(* PLC project Sin nombre, Desconocido Sin nombre 1 *)
(* stored: creationDateTime 2025-10-27T12:46:01, modificationDateTime 2025-10-27T17:09:16 *)

PROGRAM program0
  VAR
    SensorInclinacion AT %IX0.1 : BOOL;
    SensorFuego AT %IW0 : INT;
    LedAzul AT %QX0.3 : BOOL := FALSE;
    LedParacaidas AT %QX0.4 : BOOL := FALSE;
    LedRojo AT %QX0.1 : BOOL := FALSE;
  END_VAR
  VAR
    EstadoTurbulento : BOOL := FALSE;
    EstadoSobrecalentamiento : BOOL := FALSE;
  END_VAR
  VAR
    LedVerde AT %QX0.2 : BOOL := TRUE;
  END_VAR
  VAR
    EstadoSeguro : BOOL := TRUE;
    UmbralFuego : INT := 1;
    RetardoParacaidas : TIME := T#5000ms;
    Titilo : TIME := T#10ms;
    TiempoSubidaBajada : TIME := T#30000ms;
    RetardoEyeccion : TON;
    AscensoDescenso : TOF;
    ParpadeoLuces : TP;
    Despliegue : TP;
    BiestableAscDesc : RS;
  END_VAR
  VAR  (* added by the conversion: wires and edge detectors of the diagram *)
    _AND42_OUT : BOOL;
    _GT10_OUT : BOOL;
    _AND14_OUT : BOOL;
  END_VAR

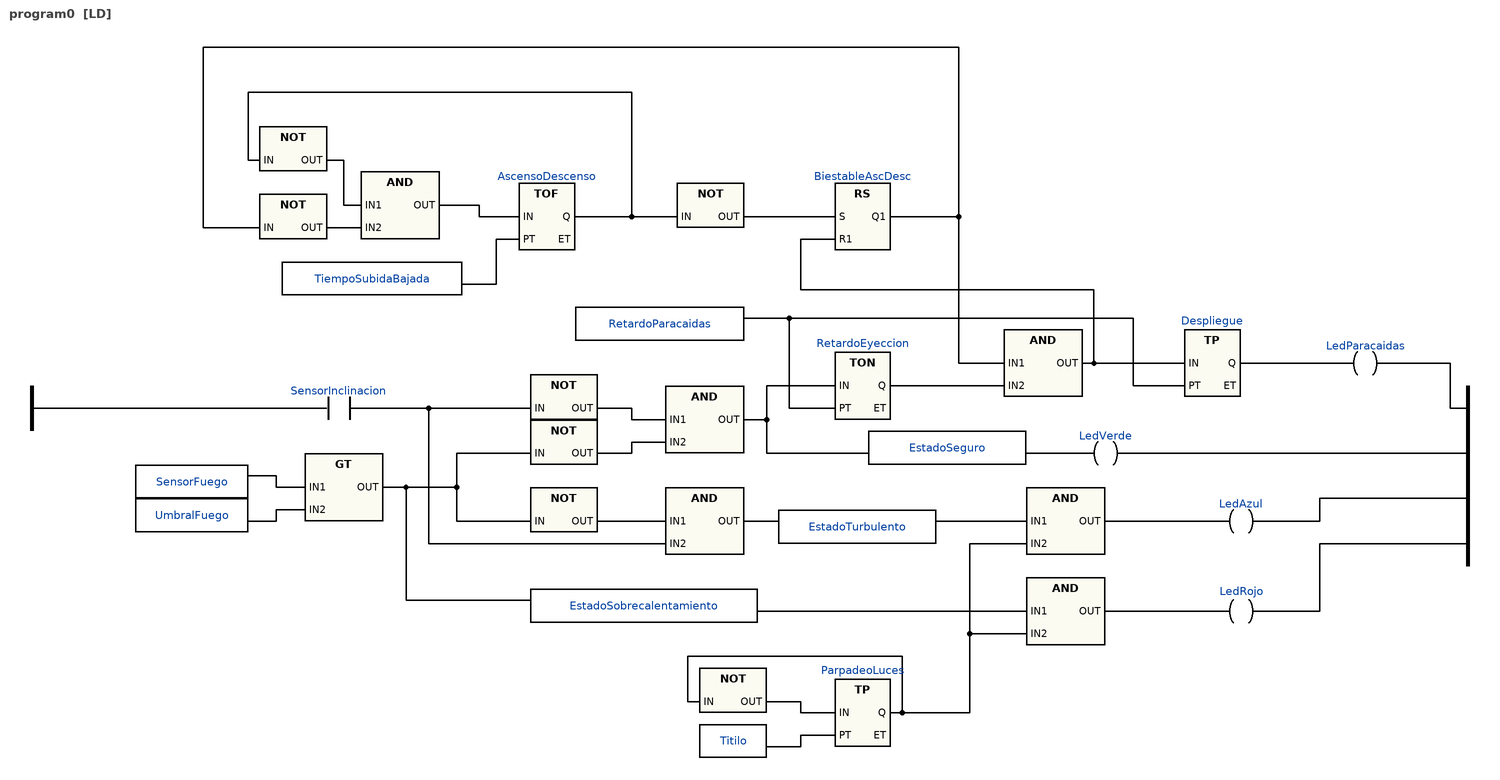
(* LD diagram, written out as Structured Text *)
AscensoDescenso(IN := NOT AscensoDescenso.Q AND NOT BiestableAscDesc.Q1, PT := TiempoSubidaBajada);
BiestableAscDesc(S := NOT AscensoDescenso.Q, R1 := _AND42_OUT);
_GT10_OUT := SensorFuego > UmbralFuego;
_AND14_OUT := NOT SensorInclinacion AND NOT _GT10_OUT;
RetardoEyeccion(IN := _AND14_OUT, PT := RetardoParacaidas);
_AND42_OUT := BiestableAscDesc.Q1 AND RetardoEyeccion.Q;
Despliegue(IN := _AND42_OUT, PT := RetardoParacaidas);
LedParacaidas := Despliegue.Q;
LedVerde := EstadoSeguro;
ParpadeoLuces(IN := NOT ParpadeoLuces.Q, PT := Titilo);
LedAzul := EstadoTurbulento AND ParpadeoLuces.Q;
LedRojo := EstadoSobrecalentamiento AND ParpadeoLuces.Q;
EstadoSeguro := _AND14_OUT;
EstadoTurbulento := NOT _GT10_OUT AND SensorInclinacion;
EstadoSobrecalentamiento := _GT10_OUT;
END_PROGRAM

CONFIGURATION Config0
  RESOURCE Res0 ON PLC
    TASK task0(INTERVAL := T#20ms, PRIORITY := 0);
    PROGRAM instance0 WITH task0 : program0;
  END_RESOURCE
END_CONFIGURATION
